(* IEC 61131-3 sources: netRob/Hardwareadapter/parser/ASCII/functions, 3 files *)

(* ---- AsciiChar.ST ---- *)
(*@PROPERTIES_EX@
TYPE: POU
LOCALE: 0
IEC_LANGUAGE: ST
PLC_TYPE: independent
PROC_TYPE: independent
*)
(*@KEY@:DESCRIPTION*)

(*@KEY@:END_DESCRIPTION*)
FUNCTION AsciiChar : STRING1
VAR_INPUT
	character: BYTE;
END_VAR
VAR
END_VAR

(*@KEY@: WORKSHEET
NAME: AsciiChar
IEC_LANGUAGE: ST
*)
CASE character OF
	000: AsciiChar := '$00';
	001: AsciiChar := '$01';
	002: AsciiChar := '$02';
	003: AsciiChar := '$03';
	004: AsciiChar := '$04';
	005: AsciiChar := '$05';
	006: AsciiChar := '$06';
	007: AsciiChar := '$07';
	008: AsciiChar := '$08';
	009: AsciiChar := '$09';
	010: AsciiChar := '$0a';
	011: AsciiChar := '$0b';
	012: AsciiChar := '$0c';
	013: AsciiChar := '$0d';
	014: AsciiChar := '$0e';
	015: AsciiChar := '$0f';
	016: AsciiChar := '$10';
	017: AsciiChar := '$11';
	018: AsciiChar := '$12';
	019: AsciiChar := '$13';
	020: AsciiChar := '$14';
	021: AsciiChar := '$15';
	022: AsciiChar := '$16';
	023: AsciiChar := '$17';
	024: AsciiChar := '$18';
	025: AsciiChar := '$19';
	026: AsciiChar := '$1a';
	027: AsciiChar := '$1b';
	028: AsciiChar := '$1c';
	029: AsciiChar := '$1d';
	030: AsciiChar := '$1e';
	031: AsciiChar := '$1f';
	032: AsciiChar := '$20';
	033: AsciiChar := '$21';
	034: AsciiChar := '$22';
	035: AsciiChar := '$23';
	036: AsciiChar := '$24';
	037: AsciiChar := '$25';
	038: AsciiChar := '$26';
	039: AsciiChar := '$27';
	040: AsciiChar := '$28';
	041: AsciiChar := '$29';
	042: AsciiChar := '$2a';
	043: AsciiChar := '$2b';
	044: AsciiChar := '$2c';
	045: AsciiChar := '$2d';
	046: AsciiChar := '$2e';
	047: AsciiChar := '$2f';
	048: AsciiChar := '$30';
	049: AsciiChar := '$31';
	050: AsciiChar := '$32';
	051: AsciiChar := '$33';
	052: AsciiChar := '$34';
	053: AsciiChar := '$35';
	054: AsciiChar := '$36';
	055: AsciiChar := '$37';
	056: AsciiChar := '$38';
	057: AsciiChar := '$39';
	058: AsciiChar := '$3a';
	059: AsciiChar := '$3b';
	060: AsciiChar := '$3c';
	061: AsciiChar := '$3d';
	062: AsciiChar := '$3e';
	063: AsciiChar := '$3f';
	064: AsciiChar := '$40';
	065: AsciiChar := '$41';
	066: AsciiChar := '$42';
	067: AsciiChar := '$43';
	068: AsciiChar := '$44';
	069: AsciiChar := '$45';
	070: AsciiChar := '$46';
	071: AsciiChar := '$47';
	072: AsciiChar := '$48';
	073: AsciiChar := '$49';
	074: AsciiChar := '$4a';
	075: AsciiChar := '$4b';
	076: AsciiChar := '$4c';
	077: AsciiChar := '$4d';
	078: AsciiChar := '$4e';
	079: AsciiChar := '$4f';
	080: AsciiChar := '$50';
	081: AsciiChar := '$51';
	082: AsciiChar := '$52';
	083: AsciiChar := '$53';
	084: AsciiChar := '$54';
	085: AsciiChar := '$55';
	086: AsciiChar := '$56';
	087: AsciiChar := '$57';
	088: AsciiChar := '$58';
	089: AsciiChar := '$59';
	090: AsciiChar := '$5a';
	091: AsciiChar := '$5b';
	092: AsciiChar := '$5c';
	093: AsciiChar := '$5d';
	094: AsciiChar := '$5e';
	095: AsciiChar := '$5f';
	096: AsciiChar := '$60';
	097: AsciiChar := '$61';
	098: AsciiChar := '$62';
	099: AsciiChar := '$63';
	100: AsciiChar := '$64';
	101: AsciiChar := '$65';
	102: AsciiChar := '$66';
	103: AsciiChar := '$67';
	104: AsciiChar := '$68';
	105: AsciiChar := '$69';
	106: AsciiChar := '$6a';
	107: AsciiChar := '$6b';
	108: AsciiChar := '$6c';
	109: AsciiChar := '$6d';
	110: AsciiChar := '$6e';
	111: AsciiChar := '$6f';
	112: AsciiChar := '$70';
	113: AsciiChar := '$71';
	114: AsciiChar := '$72';
	115: AsciiChar := '$73';
	116: AsciiChar := '$74';
	117: AsciiChar := '$75';
	118: AsciiChar := '$76';
	119: AsciiChar := '$77';
	120: AsciiChar := '$78';
	121: AsciiChar := '$79';
	122: AsciiChar := '$7a';
	123: AsciiChar := '$7b';
	124: AsciiChar := '$7c';
	125: AsciiChar := '$7d';
	126: AsciiChar := '$7e';
	127: AsciiChar := '$7f';
END_CASE;

(*@KEY@: END_WORKSHEET *)
END_FUNCTION

(* ---- InitAscii.ST ---- *)
(*@PROPERTIES_EX@
TYPE: POU
LOCALE: 0
IEC_LANGUAGE: ST
PLC_TYPE: independent
PROC_TYPE: independent
*)
(*@KEY@:DESCRIPTION*)

(*@KEY@:END_DESCRIPTION*)
FUNCTION InitAscii : BOOL
VAR_INPUT
	input: BOOL; (* ignored *)
END_VAR
VAR_EXTERNAL
	Ascii: AsciiConstants;
END_VAR

(*@KEY@: WORKSHEET
NAME: InitAscii
IEC_LANGUAGE: ST
*)
Ascii.NULL := 0;
Ascii.SOH := 1;
Ascii.STX := 2;
Ascii.ETX := 3;
Ascii.EOT := 4;
Ascii.ENQ := 5;
Ascii.ACK := 6;
Ascii.BELL := 7;
Ascii.BACKSPACE := 8;
Ascii.HORIZONTAL_TAB := 9;
Ascii.NEW_LINE := 10;
Ascii.VERTICAL_TAB := 11;
Ascii.FORMFEED := 12;
Ascii.CARRIAGE_RETURN := 13;
Ascii.SO := 14;
Ascii.SI := 15;
Ascii.DLE := 16;
Ascii.DC1 := 17;
Ascii.DC2 := 18;
Ascii.DC3 := 19;
Ascii.DC4 := 20;
Ascii.NAK := 21;
Ascii.SYN := 22;
Ascii.ETB := 23;
Ascii.CAN := 24;
Ascii.EM := 25;
Ascii.SUBSTITUDE := 26;
Ascii.ESC := 27;
Ascii.FS := 28;
Ascii.GS := 29;
Ascii.RS := 30;
Ascii.US := 31;
Ascii.SPACE := 32;
Ascii.BANG := 33;
Ascii.DOUBLE_QUOTE := 34;
Ascii.HASH := 35;
Ascii.DOLLAR := 36;
Ascii.PERCENT := 37;
Ascii.AMPERSAND := 38;
Ascii.SINGLE_QUOTE := 39;
Ascii.OPEN_PAREN := 40;
Ascii.CLOSE_PAREN := 41;
Ascii.STAR := 42;
Ascii.PLUS := 43;
Ascii.COMMA := 44;
Ascii.MINUS := 45;
Ascii.DOT := 46;
Ascii.SLASH := 47;
Ascii.NUMBER_0 := 48;
Ascii.NUMBER_1 := 49;
Ascii.NUMBER_2 := 50;
Ascii.NUMBER_3 := 51;
Ascii.NUMBER_4 := 52;
Ascii.NUMBER_5 := 53;
Ascii.NUMBER_6 := 54;
Ascii.NUMBER_7 := 55;
Ascii.NUMBER_8 := 56;
Ascii.NUMBER_9 := 57;
Ascii.COLON := 58;
Ascii.SEMICOLON := 59;
Ascii.LESS_THAN := 60;
Ascii.EQUALS := 61;
Ascii.GREATER_THAN := 62;
Ascii.QUESTION := 63;
Ascii.AT_SIGN := 64;
Ascii.UPPERCASE_A := 65;
Ascii.UPPERCASE_B := 66;
Ascii.UPPERCASE_C := 67;
Ascii.UPPERCASE_D := 68;
Ascii.UPPERCASE_E := 69;
Ascii.UPPERCASE_F := 70;
Ascii.UPPERCASE_G := 71;
Ascii.UPPERCASE_H := 72;
Ascii.UPPERCASE_I := 73;
Ascii.UPPERCASE_J := 74;
Ascii.UPPERCASE_K := 75;
Ascii.UPPERCASE_L := 76;
Ascii.UPPERCASE_M := 77;
Ascii.UPPERCASE_N := 78;
Ascii.UPPERCASE_O := 79;
Ascii.UPPERCASE_P := 80;
Ascii.UPPERCASE_Q := 81;
Ascii.UPPERCASE_R := 82;
Ascii.UPPERCASE_S := 83;
Ascii.UPPERCASE_T := 84;
Ascii.UPPERCASE_U := 85;
Ascii.UPPERCASE_V := 86;
Ascii.UPPERCASE_W := 87;
Ascii.UPPERCASE_X := 88;
Ascii.UPPERCASE_Y := 89;
Ascii.UPPERCASE_Z := 90;
Ascii.OPEN_BRACKET := 91;
Ascii.BACKSLASH := 92;
Ascii.CLOSE_BRACKET := 93;
Ascii.CARET := 94;
Ascii.UNDERSCORE := 95;
Ascii.BACKQUOTE := 96;
Ascii.LOWERCASE_A := 97;
Ascii.LOWERCASE_B := 98;
Ascii.LOWERCASE_C := 99;
Ascii.LOWERCASE_D := 100;
Ascii.LOWERCASE_E := 101;
Ascii.LOWERCASE_F := 102;
Ascii.LOWERCASE_G := 103;
Ascii.LOWERCASE_H := 104;
Ascii.LOWERCASE_I := 105;
Ascii.LOWERCASE_J := 106;
Ascii.LOWERCASE_K := 107;
Ascii.LOWERCASE_L := 108;
Ascii.LOWERCASE_M := 109;
Ascii.LOWERCASE_N := 110;
Ascii.LOWERCASE_O := 111;
Ascii.LOWERCASE_P := 112;
Ascii.LOWERCASE_Q := 113;
Ascii.LOWERCASE_R := 114;
Ascii.LOWERCASE_S := 115;
Ascii.LOWERCASE_T := 116;
Ascii.LOWERCASE_U := 117;
Ascii.LOWERCASE_V := 118;
Ascii.LOWERCASE_W := 119;
Ascii.LOWERCASE_X := 120;
Ascii.LOWERCASE_Y := 121;
Ascii.LOWERCASE_Z := 122;
Ascii.OPEN_BRACE := 123;
Ascii.PIPE := 124;
Ascii.CLOSE_BRACE := 125;
Ascii.TILDE := 126;
Ascii.DELETE := 127;

InitAscii := input;

(*@KEY@: END_WORKSHEET *)
END_FUNCTION

(* ---- ReadBuffer.ST ---- *)
(*@PROPERTIES_EX@
TYPE: POU
LOCALE: 0
IEC_LANGUAGE: ST
PLC_TYPE: independent
PROC_TYPE: independent
*)
(*@KEY@:DESCRIPTION*)

(*@KEY@:END_DESCRIPTION*)
FUNCTION_BLOCK ReadBuffer
VAR_INPUT
	buffer: OSCAT_NETWORK.NW_BUF_LONG;
END_VAR
VAR_OUTPUT
	actualCharacter: BYTE;
END_VAR
VAR
	position: DINT := 0;
END_VAR
VAR_EXTERNAL
	Constants: GeneralConstants;
	Ascii: AsciiConstants;
	Json: JsonConstants;
END_VAR

(*@KEY@: WORKSHEET
NAME: ReadBuffer
IEC_LANGUAGE: ST
*)
(* Initialise position to the begin of the buffer or *)
(* Reset position to the begin of a (probably new) buffer *)
IF ParserGlobals.resetParser THEN
	position := DINT#0;
	actualCharacter := BYTE#0;
	RETURN;
END_IF;
(* Get the actual character and shift position if it isn't the end *)
actualCharacter := buffer[position];
IF NOT(actualCharacter = Ascii.NULL) THEN
	position := position +1;
END_IF;

(*@KEY@: END_WORKSHEET *)
END_FUNCTION_BLOCK
